Staubli VAL3: matrix.dtx

mdesc mNomSpeed
num nMatrix1[3 4]
num nMatrix2[3 4]
num nResult[1 1]
